Universal Robots PolyScope program: pickandplace.urp

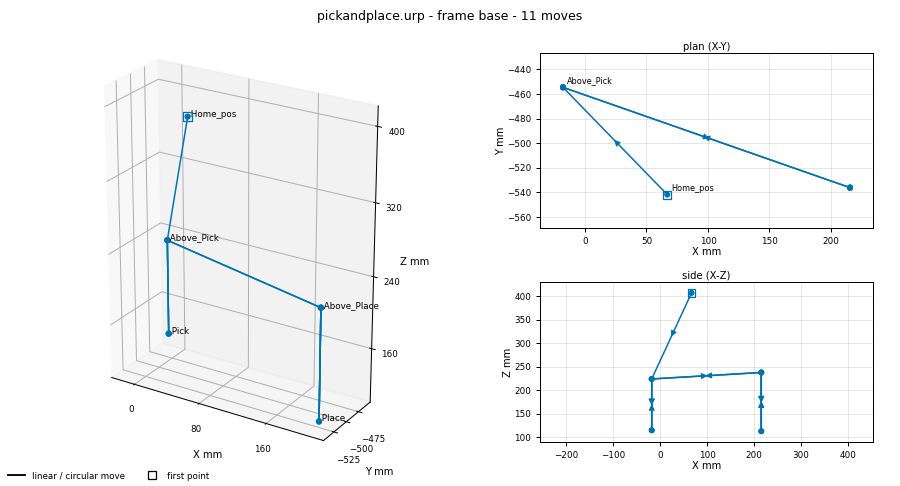
[picture p0: tool path of pickandplace.urp in frame base, 11 of 12 moves have a stored position in this frame; points joined in program order, loops and branches not executed]
Program pickandplace (installation=default directory=/programs/RemoteOperation createdIn=5.10.0.106268 lastSavedIn=5.10.0.106268 robotSerialNumber=20185500191)
Calibrated DH parameters: a=[0.000131, -0.165639, -0.102041, 0.000082, 0.000046, 0]; d=[0.162455, 220.258006, 1988.136334, -2208.260978, 0.099826, 0.099896]; alpha=[1.570482, -0.001777, -0.000172, 1.570393, -1.570735, 0]; deltaTheta=[0, -1.170526, -0.137148, 1.307669, -0.000001, 0]
Robot Program (runOnlyOnce=false)
  MoveJ speed 60 deg/s, acceleration 80 deg/s^2 (useActiveTCP=true) feature=Base
    Waypoint Autostart (Relative): relativeFromPosition TCP in base x=-17.861 y=-454.579 z=157.55 mm, rx=2.1915 ry=2.2509 rz=-0.0001 rad; joints [-75.231, -86.581, -116.729, -66.688, 89.927, 103.249] deg; TCP offset x=0 y=0 z=174 mm, rx=0 ry=0 rz=0 rad; TCP in base x=-17.86 y=-454.578 z=157.54 mm, rx=2.1915 ry=2.2509 rz=-0.0001 rad; joints [-75.231, -86.581, -116.731, -66.685, 89.928, 103.25] deg
    Waypoint Home_pos: TCP in base x=66.883 y=-541.756 z=407.399 mm, rx=2.1915 ry=2.2509 rz=-0.0001 rad; joints [-68.794, -96.625, -69.103, -104.273, 89.914, 109.67] deg
  MoveL speed 250 mm/s, acceleration 1200 mm/s^2 (useActiveTCP=true) feature=Base
    Waypoint Above_Pick: motionParameters(blendRadius=0.05); TCP in base x=-17.886 y=-454.566 z=224.166 mm, rx=-2.1915 ry=-2.2509 rz=0.0001 rad; joints [-75.228, -83.558, -109.209, -77.235, 89.926, 103.256] deg
    Waypoint Pick: TCP in base x=-17.859 y=-454.546 z=114.83 mm, rx=2.1915 ry=2.2509 rz=0 rad; joints [-75.232, -89.551, -120.878, -59.573, 89.929, 103.244] deg
    'Close gripper command should be inserted here'
    Wait Sleep waitTime=1
    SetPayload (workpieceName=PartInHand)
    Waypoint Above_Pick: motionParameters(blendRadius=0.05); TCP in base x=-17.886 y=-454.566 z=224.166 mm, rx=-2.1915 ry=-2.2509 rz=0.0001 rad; joints [-75.228, -83.558, -109.209, -77.235, 89.926, 103.256] deg
    Waypoint Above_Place: motionParameters(blendRadius=0.05); TCP in base x=215.486 y=-536.12 z=237.921 mm, rx=2.1915 ry=2.2509 rz=-0.0001 rad; joints [-54.751, -100.29, -89.806, -79.902, 89.915, 123.707] deg
    Waypoint Place: TCP in base x=215.472 y=-536.096 z=112.892 mm, rx=-2.1915 ry=-2.251 rz=0.0001 rad; joints [-54.758, -105.835, -102.217, -61.952, 89.917, 123.688] deg
    'Open gripper command should be inserted here'
    Wait Sleep waitTime=1
    SetPayload (workpieceName=Gripper)
    Waypoint Above_Place: TCP in base x=215.486 y=-536.12 z=237.921 mm, rx=2.1915 ry=2.2509 rz=-0.0001 rad; joints [-54.751, -100.29, -89.806, -79.902, 89.915, 123.707] deg
    Waypoint Place: TCP in base x=215.472 y=-536.096 z=112.892 mm, rx=-2.1915 ry=-2.251 rz=0.0001 rad; joints [-54.758, -105.835, -102.217, -61.952, 89.917, 123.688] deg
    'Close gripper command should be inserted here'
    Wait Sleep waitTime=1
    SetPayload (workpieceName=PartInHand)
    Waypoint Above_Place: motionParameters(blendRadius=0.05); TCP in base x=215.486 y=-536.12 z=237.921 mm, rx=2.1915 ry=2.2509 rz=-0.0001 rad; joints [-54.751, -100.29, -89.806, -79.902, 89.915, 123.707] deg
    Waypoint Above_Pick: motionParameters(blendRadius=0.05); TCP in base x=-17.886 y=-454.566 z=224.166 mm, rx=-2.1915 ry=-2.2509 rz=0.0001 rad; joints [-75.228, -83.558, -109.209, -77.235, 89.926, 103.256] deg
    Waypoint Pick: TCP in base x=-17.859 y=-454.546 z=114.83 mm, rx=2.1915 ry=2.2509 rz=0 rad; joints [-75.232, -89.551, -120.878, -59.573, 89.929, 103.244] deg
    'Open gripper command should be inserted here'
    Wait Sleep waitTime=1
